TYPE DUT_SIMULATION :
STRUCT
XPosition0 : LREAL;
XPosition1 : lreal;
XPosition2 : lreal;
XPosition3 : lreal;
XPosition4 : lreal;
XPosition5 : lreal;
XPosition6 : lreal;
XPosition7 : lreal;
XPosition8 : lreal;
XPosition9 : lreal;
XPosition10 :LREAL;

Cocktail			: DUT_SIMU_SKILLSTATE;
Cookie				: DUT_SIMU_SKILLSTATE;
Topping_Beckhoff	: DUT_SIMU_SKILLSTATE;
Topping_Bosch		: DUT_SIMU_SKILLSTATE;

END_STRUCT
END_TYPE

(* stored: Version 1.1.0.1, ProductVersion 3.1.0.25
   DUT DUT_SIMULATION: Id {4c50ade2-26f4-4662-b1fd-9ae8096ff500} *)
